FUNCTION_BLOCK FB_Axis
VAR_INPUT
	sName:STRING;
	Axis:Axis_ref;
	bEnable:BOOL:=FALSE;
	bHalt:BOOL:=FALSE;
	bHome:BOOL:=FALSE;
	bReset:BOOL:=FALSE;
	bSetPosition:BOOL:=FALSE;
	Dist:REAL;
	bMoveRel:BOOL:=FALSE;
	bMoveRelBusy:BOOL;
	rPos:LREAL;
	rVel:LREAL;
	rAcc:LREAL;
	rDec:LREAL;
	jJerk:LREAL;
	bMoveABS:BOOL:=FALSE;
	bMoveAbsBusy:BOOL;
	bJogPos:BOOL;
	bJogNeg:BOOL;
	rStep: REAL:=400;
	rStep_vel: REAL:=400;
	bmanual:BOOL:=FALSE;
	bDo_Step_FW:BOOL:=FALSE;
	bDo_Step_BW:BOOL:=FALSE;
	stepFW_state:INT:=0;
	stepBW_state:INT:=0;
	bStop:BOOL:=0;
	bHomeBusy:BOOL;
	ton_Reset: TON;
END_VAR

VAR_OUTPUT
	bBusy: BOOL;
	bError:BOOL;
	bInPos:BOOL;
	rActPos:LREAL;
	rActVel:LREAL;
	bRelDone:BOOL;
	bAbsDone:BOOL;
END_VAR
VAR
	tDelay: TON;
	bDelay:BOOL:=FALSE;
	MoveAbsolute: MC_MoveAbsolute;
	power: MC_Power;
	Reset: MC_Reset;
	SetPosition: MC_SetPosition;
	JOG: MC_Jog;
	RELATIVE: MC_MoveRelative;
	HALT: MC_Halt;
	HOME: MC_Home;
	bFirst_run:BOOL:=FALSE;
	bStopBusy:BOOL;
	
	
	
	
END_VAR

IF NOT bFirst_run THEN
	RESET.Execute:=TRUE;
END_IF


rActPos:=Axis.NcToPlc.ActPos;
rActVel:=Axis.NcToPlc.ActVelo;

STEP_FW();


IF RELATIVE.Busy OR JOG.Busy OR moveAbsolute.busy THEN
	bBusy:=TRUE;
ELSE
	bBusy:=FALSE;
END_IF

IF POWER.error OR RELATIVE.error OR MoveAbsolute.error OR JOG.error THEN
	bError:=TRUE;
ELSE
	bError:=FALSE;
END_IF

IF RELATIVE.Done OR JOG.Done OR moveAbsolute.Done THEN
	bInPos:=TRUE;
ELSE
	bInPos:=FALSE;
END_IF
motion_commands();
(*
RELATIVE(
	Axis:= Axis, 
	Execute:=bMoveRel , 
	Distance:= Dist, 
	Velocity:=rVel , 
	Acceleration:= , 
	Deceleration:= , 
	Jerk:= , 
	BufferMode:= , 
	Options:= , 
	Done=> bRelDone, 
	Busy=> , 
	Active=> , 
	CommandAborted=> , 
	Error=> , 
	ErrorID=> );
	
JOG(
	Axis:=Axis , 
	JogForward:= bJogPos, 
	JogBackwards:=bJogNeg , 
	Mode:= E_JogMode.MC_JOGMODE_CONTINOUS,
	Position:=rPos , 
	Velocity:= rVel, 
	Acceleration:= , 
	Deceleration:= , 
	Jerk:= , 
	Done=> , 
	Busy=> , 
	Active=> , 
	CommandAborted=> , 
	Error=> , 
	ErrorID=> );

Power(
	Axis:= Axis, 
	Enable:= bEnable, 
	Enable_Positive:= bEnable, 
	Enable_Negative:= bEnable, 
	Override:= 100, 
	BufferMode:= , 
	Options:= , 
	Status=> , 
	Busy=> , 
	Active=> , 
	Error=> , 
	ErrorID=> );

Reset(
	Axis:= Axis, 
	Execute:= bReset, 
	Done=> , 
	Busy=> , 
	Error=> , 
	ErrorID=> );
	
SetPosition(
	Axis:= Axis, 
	Execute:= bSetPosition, 
	Position:= rPos, 
	Mode:= , 
	Options:= , 
	Done=> , 
	Busy=> , 
	Error=> , 
	ErrorID=> );

MoveAbsolute(
	Axis:= Axis, 
	Execute:= bMoveABS, 
	Position:= rPos, 
	Velocity:= rVel, 
	Acceleration:= , 
	Deceleration:= , 
	Jerk:= , 
	BufferMode:= , 
	Options:= , 
	Done=> bAbsDone, 
	Busy=> , 
	Active=> , 
	CommandAborted=> , 
	Error=> , 
	ErrorID=> );
	
HALT(
	Axis:= Axis, 
	Execute:= bHalt, 
	Deceleration:= , 
	Jerk:= , 
	BufferMode:= , 
	Options:= , 
	Done=> , 
	Busy=> , 
	Active=> , 
	CommandAborted=> , 
	Error=> , 
	ErrorID=> );

	*)

METHOD clear_cmd_req : BOOL
VAR_INPUT
END_VAR

bMoveABS:= bMoveRel:= bJogPos:= bJogNeg:=FALSE;
END_METHOD

ACTION motion_commands:
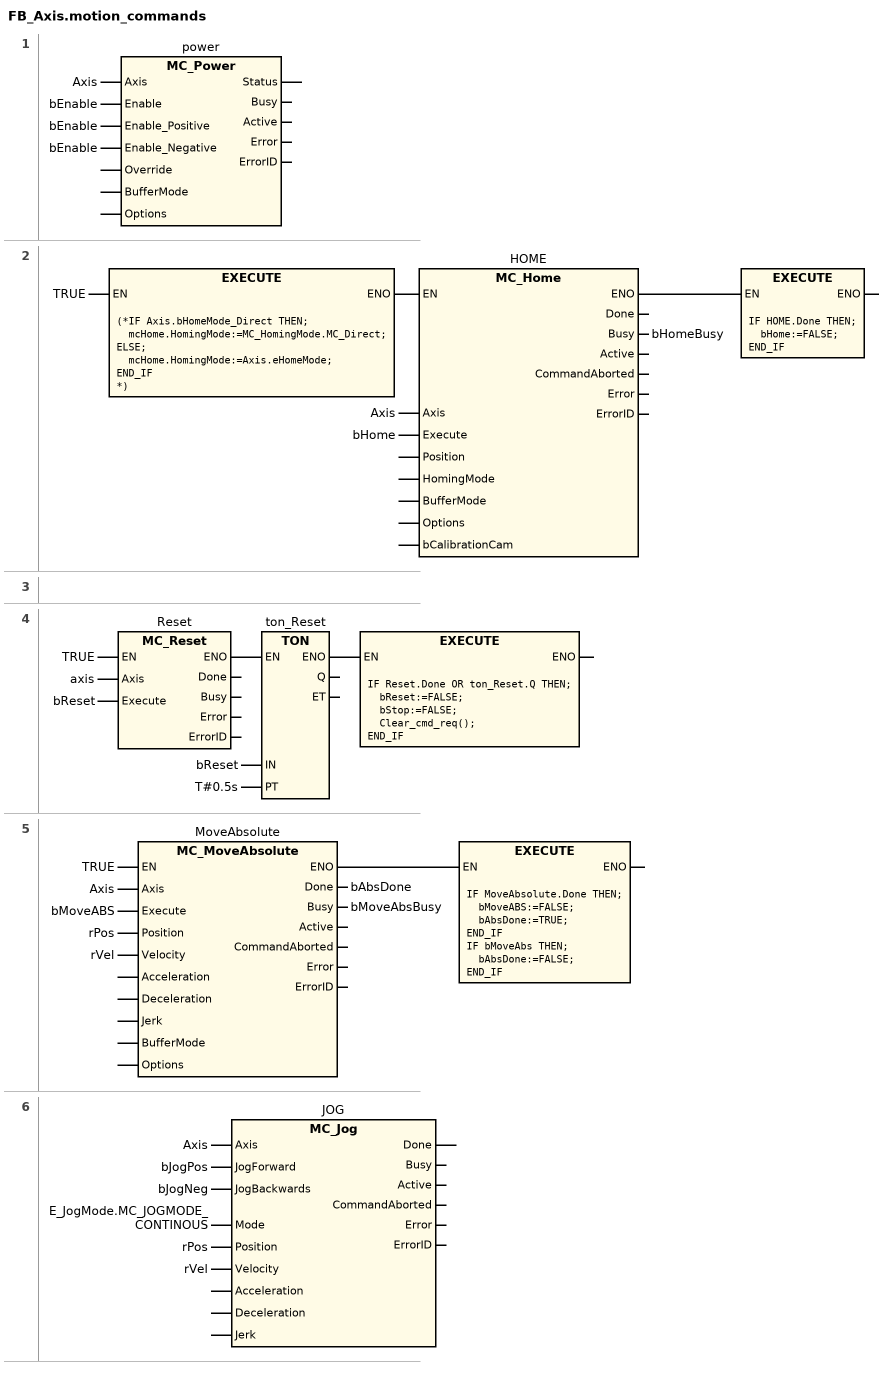
// NETWORK 1
power(Axis := Axis, Enable := bEnable, Enable_Positive := bEnable, Enable_Negative := bEnable); // MC_Power

// NETWORK 2

(*IF Axis.bHomeMode_Direct THEN;
	mcHome.HomingMode:=MC_HomingMode.MC_Direct;
ELSE;
	mcHome.HomingMode:=Axis.eHomeMode;
END_IF
*)
HOME(Axis := Axis, Execute := bHome, Busy => bHomeBusy); // MC_Home

IF HOME.Done THEN;
	bHome:=FALSE;
END_IF

// NETWORK 3

// NETWORK 4
Reset(Axis := axis, Execute := bReset); // MC_Reset
ton_Reset(IN := bReset, PT := T#0.5s); // TON

IF Reset.Done OR ton_Reset.Q THEN;
	bReset:=FALSE;
	bStop:=FALSE;
	Clear_cmd_req();
END_IF

// NETWORK 5
MoveAbsolute(
    Axis := Axis,
    Execute := bMoveABS,
    Position := rPos,
    Velocity := rVel,
    Done => bAbsDone,
    Busy => bMoveAbsBusy); // MC_MoveAbsolute

IF MoveAbsolute.Done THEN;
	bMoveABS:=FALSE;
	bAbsDone:=TRUE;
END_IF
IF bMoveAbs THEN;
	bAbsDone:=FALSE;
END_IF

// NETWORK 6
JOG(
    Axis := Axis,
    JogForward := bJogPos,
    JogBackwards := bJogNeg,
    Mode := E_JogMode.MC_JOGMODE_CONTINOUS,
    Position := rPos,
    Velocity := rVel); // MC_Jog

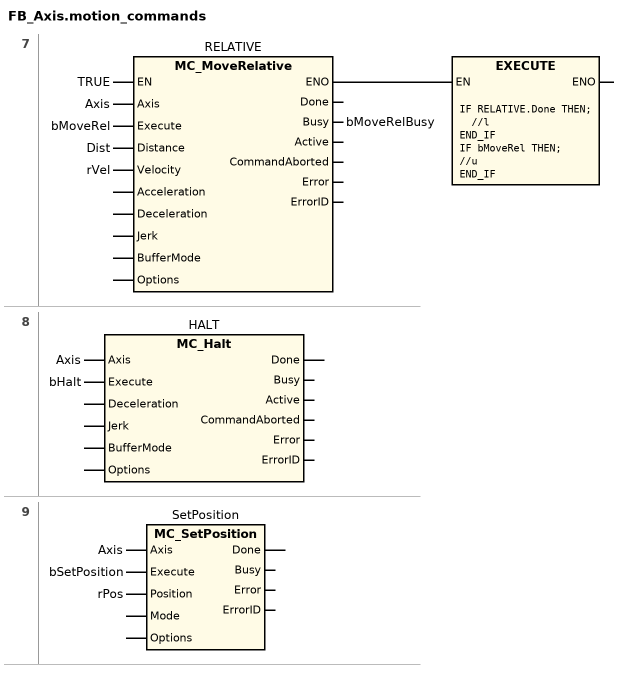
// NETWORK 7
RELATIVE(Axis := Axis, Execute := bMoveRel, Distance := Dist, Velocity := rVel, Busy => bMoveRelBusy); // MC_MoveRelative

IF RELATIVE.Done THEN;
	//l
END_IF
IF bMoveRel THEN;
//u
END_IF

// NETWORK 8
HALT(Axis := Axis, Execute := bHalt); // MC_Halt

// NETWORK 9
SetPosition(Axis := Axis, Execute := bSetPosition, Position := rPos); // MC_SetPosition
END_ACTION

METHOD STEP_FW : BOOL
VAR_INPUT
END_VAR
 
CASE stepFW_state OF
	
	0:
	IF bDo_Step_FW AND NOT bManual THEN		
		bMoveRel:=FALSE;
		//bReset:=TRUE;
		bDo_Step_FW:=FALSE;
		stepFW_state := 1;	
	END_IF

	1:
	Dist:=rStep;
	rVel:=rStep_Vel;
	bEnable:=TRUE;
	bMoveRel:=FALSE;
	stepFW_state := 2;
	//bReset:=FALSE;
	
	2:
	bMoveRel:=TRUE;
	stepFW_state := 3;
	
	3:
	IF RELATIVE.Done THEN
		 bDo_Step_FW:=FALSE;
		 stepFW_state := 0;
	END_IF
	
	
	
	
END_CASE
END_METHOD

END_FUNCTION_BLOCK

(* stored: Version 1.1.0.1, ProductVersion 3.1.4024.12
   POU FB_Axis: Id {1ec8daca-b967-496e-b296-4221933406bb}, SpecialFunc None
   Method clear_cmd_req: Id {c115c33f-8377-4dd1-8142-a1b93e7b6e59}
   Action motion_commands: Id {3ce19d79-aafb-462a-93a0-e6614d400606}
   Method STEP_FW: Id {14856ee9-0d4e-4730-ba53-d6af6d59f53f} *)
